// TIA Portal V18 export
FUNCTION_BLOCK "FB2-meteringFB"   // FB2, LAD
{ S7_Optimized_Access := 'TRUE' }
VERSION : 0.1
// stored: AutoNumber true, IsIECCheckEnabled false, IsRetainMemResEnabled false, MemoryReserve 100, SetENOAutomatically false, UDAEnableTagReadback false
   VAR_INPUT
      Metering_function : Int;
      "DO Continuous metering" : Bool;
      Dispensing_time : DInt;
      "Set Qty in ml" : Real;
      "VC1 Pulses" : DInt;
      "VC2 Pulses" : DInt;
      VC1_impulse : Real;
      VC2_impulse : Real;
      "Outlet Open  to Pump ON A delay" : DInt;
      "Outlet Open  to Pump ON B delay" : DInt;
      "Pump Off  to Inlet A Close" : DInt;
      "Pump Off  to Inlet B Close" : DInt;
      "Mixer ON to Outlet ON" : DInt;
      "Pump Off  to Outlet Close" : DInt;
      "Outlet Close to Mixer Off" : DInt;
   END_VAR
   VAR_OUTPUT
      "Volume dispensed" : Real;
      "Run time" : Int;
   END_VAR
   VAR_IN_OUT
      ON_inlet_A : Bool;
      ON_inlet_B : Bool;
      ON_Pump_A : Bool;
      ON_pump_B : Bool;
      ON_valve_A : Bool;
      ON_valve_B : Bool;
      ON_Mixer : Bool;
      "Start Metering" : Bool;
      "Stop metering" : Bool;
      "Process running" : Bool;
      "process completed" : Bool;
   END_VAR
   VAR
      "pump A to valveA delay" : Bool;
      "Pump B to valve B delay" : Bool;
      "Pump Off to mixer off delay_1" : Bool;
      "VC1 pulses prev" : DInt;
      "VC2 pulses prev" : DInt;
      "VC1 pulse generted" : DInt;
      "VC2 pulse generated" : DInt;
      "Pump A Voulme dispensed" : Real;
      "Pump B volume dispensed" : Real;
      "Total Volume dispensed" : Real;
      "metering started" : Bool;
      "metering time in msec" : DInt;
      "dispense time elapsed" : Bool;
      R_TRIG_Instance { S7_SetPoint := 'True'} : R_TRIG;
      IEC_Timer_0_Instance { S7_SetPoint := 'True'} : TON_TIME;
      IEC_Timer_0_Instance_1 { S7_SetPoint := 'True'} : TON_TIME;
      IEC_Timer_0_Instance_2 { S7_SetPoint := 'True'} : TON_TIME;
      R_TRIG_Instance_1 { S7_SetPoint := 'True'} : R_TRIG;
      temp { S7_SetPoint := 'True'} : Bool;
      IEC_Timer_0_Instance_3 { S7_SetPoint := 'True'} : TON_TIME;
      IEC_Timer_0_Instance_4 { S7_SetPoint := 'True'} : TON_TIME;
      IEC_Timer_0_Instance_5 { S7_SetPoint := 'True'} : TON_TIME;
      IEC_Timer_0_Instance_6 { S7_SetPoint := 'True'} : TON_TIME;
      IEC_Timer_0_Instance_7 { S7_SetPoint := 'True'} : TON_TIME;
      IEC_Timer_0_Instance_8 { S7_SetPoint := 'True'} : TON_TIME;
   END_VAR
   VAR_TEMP
      Ons_temp : Bool;
   END_VAR
   VAR_TEMP   // added for the SCL form of the ladder/FBD networks
      _w1 : Bool;
      _w2 : Bool;
      _w3 : Bool;
   END_VAR
BEGIN

REGION Network 1
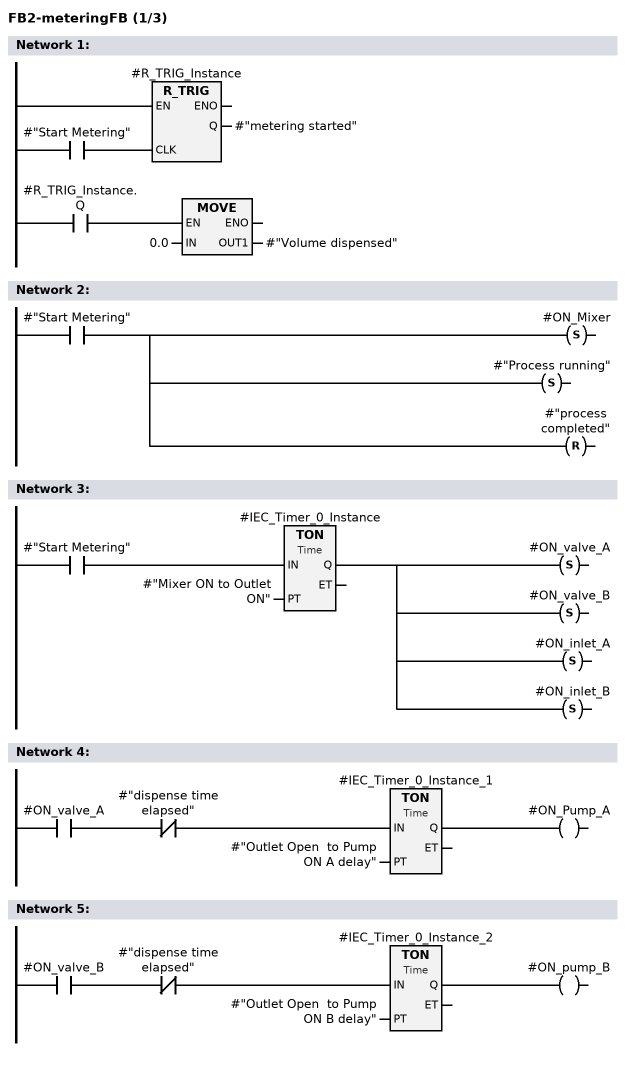
   RUNG wire#powerrail
      #R_TRIG_Instance.R_TRIG(CLK := wire#w1, Q => #"metering started")
   END_RUNG
   RUNG wire#powerrail
      Contact( #"Start Metering" )
   END_RUNG wire#w1
   RUNG wire#powerrail
      Contact( #R_TRIG_Instance.Q )
      Move(in := 0.0, out1 => #"Volume dispensed")
   END_RUNG
   // the same network as SCL:
   #R_TRIG_Instance(CLK := #"Start Metering", Q => #"metering started");   // R_TRIG
   IF #R_TRIG_Instance.Q THEN #"Volume dispensed" := 0.0; END_IF;
END_REGION

REGION Network 2
   RUNG wire#powerrail
      Contact( #"Start Metering" )
      wire#w1
      S_Coil( #ON_Mixer )
   END_RUNG
   RUNG wire#w1
      S_Coil( #"Process running" )
   END_RUNG
   RUNG wire#w1
      R_Coil( #"process completed" )
   END_RUNG
   // the same network as SCL:
   IF #"Start Metering" THEN
       #ON_Mixer := TRUE;
       #"Process running" := TRUE;
       #"process completed" := FALSE;
   END_IF;
END_REGION

REGION Network 3
   RUNG wire#powerrail
      Contact( #"Start Metering" )
      { S7_Templates := "time_type := Time" } #IEC_Timer_0_Instance.TON(pt := #"Mixer ON to Outlet ON", et =>)
      wire#w1
      S_Coil( #ON_valve_A )
   END_RUNG
   RUNG wire#w1
      S_Coil( #ON_valve_B )
   END_RUNG
   RUNG wire#w1
      S_Coil( #ON_inlet_A )
   END_RUNG
   RUNG wire#w1
      S_Coil( #ON_inlet_B )
   END_RUNG
   // the same network as SCL:
   #IEC_Timer_0_Instance(IN := #"Start Metering", PT := #"Mixer ON to Outlet ON");   // TON
   IF #IEC_Timer_0_Instance.Q THEN
       #ON_valve_A := TRUE;
       #ON_valve_B := TRUE;
       #ON_inlet_A := TRUE;
       #ON_inlet_B := TRUE;
   END_IF;
END_REGION

REGION Network 4
   RUNG wire#powerrail
      Contact( #ON_valve_A )
      I_Contact( #"dispense time elapsed" )
      { S7_Templates := "time_type := Time" } #IEC_Timer_0_Instance_1.TON(pt := #"Outlet Open  to Pump ON A delay", et =>)
      Coil( #ON_Pump_A )
   END_RUNG
   // the same network as SCL:
   #IEC_Timer_0_Instance_1(IN := #ON_valve_A AND NOT #"dispense time elapsed",   // TON
                           PT := #"Outlet Open  to Pump ON A delay");
   #ON_Pump_A := #IEC_Timer_0_Instance_1.Q;
END_REGION

REGION Network 5
   RUNG wire#powerrail
      Contact( #ON_valve_B )
      I_Contact( #"dispense time elapsed" )
      { S7_Templates := "time_type := Time" } #IEC_Timer_0_Instance_2.TON(pt := #"Outlet Open  to Pump ON B delay", et =>)
      Coil( #ON_pump_B )
   END_RUNG
   // the same network as SCL:
   #IEC_Timer_0_Instance_2(IN := #ON_valve_B AND NOT #"dispense time elapsed",   // TON
                           PT := #"Outlet Open  to Pump ON B delay");
   #ON_pump_B := #IEC_Timer_0_Instance_2.Q;
END_REGION

REGION Network 6
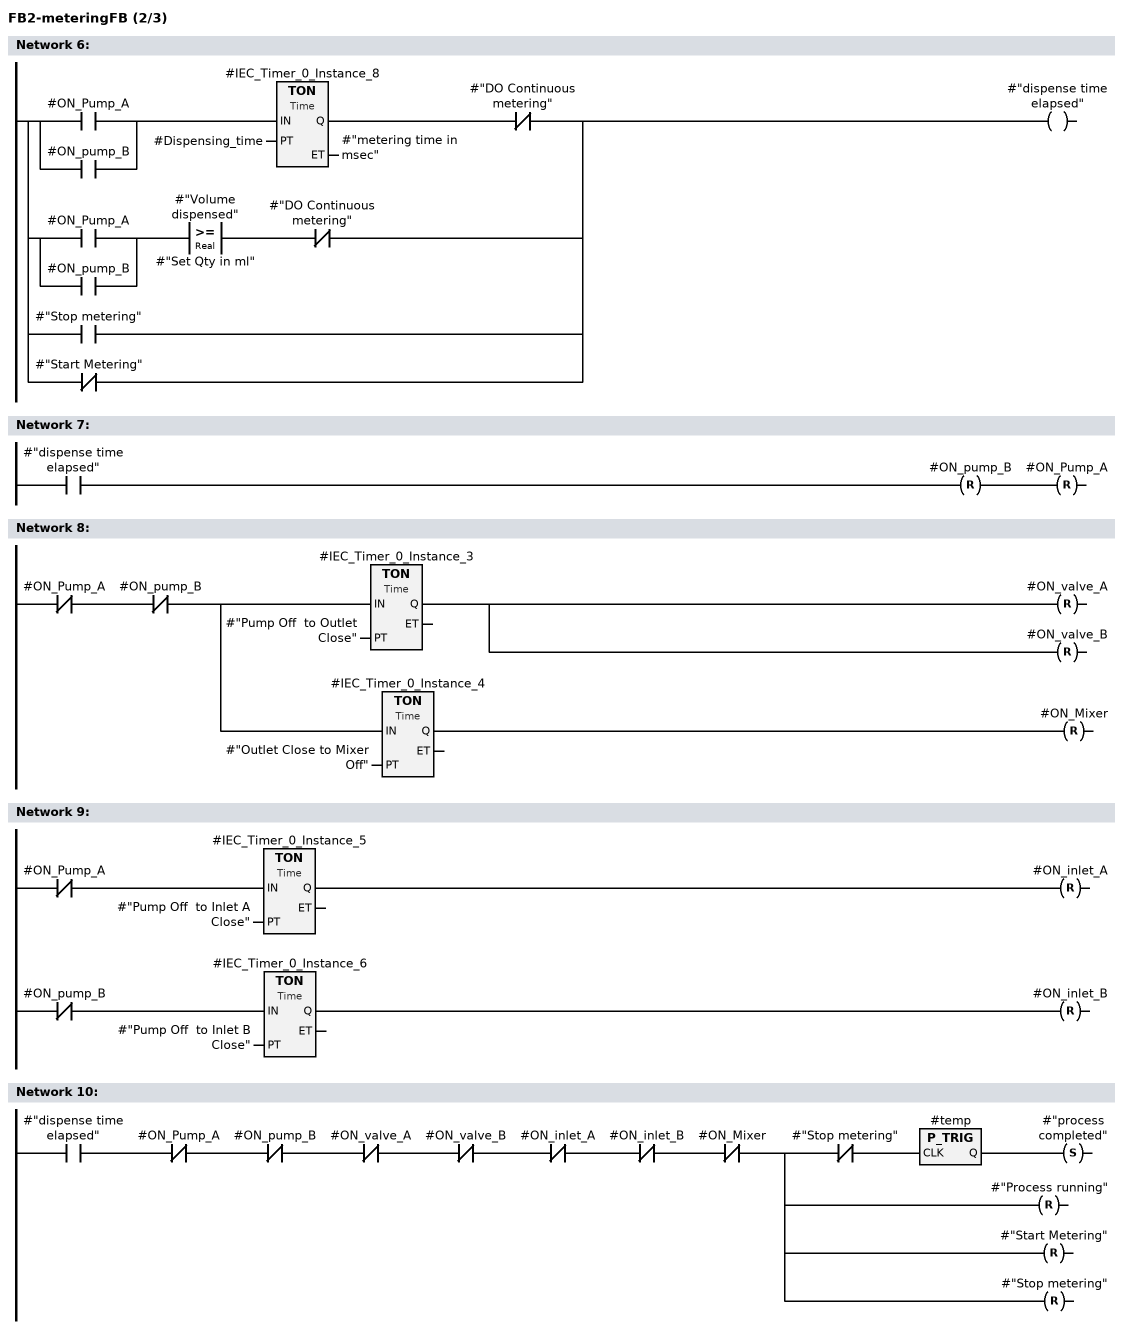
   RUNG wire#powerrail
      Contact( #ON_Pump_A )
      wire#w1
      { S7_Templates := "time_type := Time" } #IEC_Timer_0_Instance_8.TON(pt := #Dispensing_time, et => #"metering time in msec")
      I_Contact( #"DO Continuous metering" )
      wire#w2
      Coil( #"dispense time elapsed" )
   END_RUNG
   RUNG wire#powerrail
      Contact( #ON_pump_B )
   END_RUNG wire#w1
   RUNG wire#powerrail
      Contact( #ON_Pump_A )
      wire#w3
      { S7_Templates := "SrcType := Real" } GE_Contact(in1 := #"Volume dispensed", in2 := #"Set Qty in ml")
      I_Contact( #"DO Continuous metering" )
   END_RUNG wire#w2
   RUNG wire#powerrail
      Contact( #ON_pump_B )
   END_RUNG wire#w3
   RUNG wire#powerrail
      Contact( #"Stop metering" )
   END_RUNG wire#w2
   RUNG wire#powerrail
      I_Contact( #"Start Metering" )
   END_RUNG wire#w2
   // the same network as SCL:
   #IEC_Timer_0_Instance_8(IN := #ON_Pump_A OR #ON_pump_B,   // TON
                           PT := #Dispensing_time,
                           ET => #"metering time in msec");
   #"dispense time elapsed" := (#IEC_Timer_0_Instance_8.Q AND NOT #"DO Continuous metering") OR ((#ON_Pump_A OR #ON_pump_B) AND (#"Volume dispensed" >= #"Set Qty in ml") AND NOT #"DO Continuous metering") OR #"Stop metering" OR NOT #"Start Metering";
END_REGION

REGION Network 7
   RUNG wire#powerrail
      Contact( #"dispense time elapsed" )
      R_Coil( #ON_pump_B )
      R_Coil( #ON_Pump_A )
   END_RUNG
   // the same network as SCL:
   IF #"dispense time elapsed" THEN
       #ON_pump_B := FALSE;
       #ON_Pump_A := FALSE;
   END_IF;
END_REGION

REGION Network 8
   RUNG wire#powerrail
      I_Contact( #ON_Pump_A )
      I_Contact( #ON_pump_B )
      wire#w1
      { S7_Templates := "time_type := Time" } #IEC_Timer_0_Instance_3.TON(pt := #"Pump Off  to Outlet Close", et =>)
      wire#w2
      R_Coil( #ON_valve_A )
   END_RUNG
   RUNG wire#w2
      R_Coil( #ON_valve_B )
   END_RUNG
   RUNG wire#w1
      { S7_Templates := "time_type := Time" } #IEC_Timer_0_Instance_4.TON(pt := #"Outlet Close to Mixer Off", et =>)
      R_Coil( #ON_Mixer )
   END_RUNG
   // the same network as SCL:
   #_w1 := NOT #ON_Pump_A AND NOT #ON_pump_B;
   #IEC_Timer_0_Instance_3(IN := #_w1, PT := #"Pump Off  to Outlet Close");   // TON
   IF #IEC_Timer_0_Instance_3.Q THEN
       #ON_valve_A := FALSE;
       #ON_valve_B := FALSE;
   END_IF;
   #IEC_Timer_0_Instance_4(IN := #_w1, PT := #"Outlet Close to Mixer Off");   // TON
   IF #IEC_Timer_0_Instance_4.Q THEN #ON_Mixer := FALSE; END_IF;
END_REGION

REGION Network 9
   RUNG wire#powerrail
      I_Contact( #ON_Pump_A )
      { S7_Templates := "time_type := Time" } #IEC_Timer_0_Instance_5.TON(pt := #"Pump Off  to Inlet A Close", et =>)
      R_Coil( #ON_inlet_A )
   END_RUNG
   RUNG wire#powerrail
      I_Contact( #ON_pump_B )
      { S7_Templates := "time_type := Time" } #IEC_Timer_0_Instance_6.TON(pt := #"Pump Off  to Inlet B Close", et =>)
      R_Coil( #ON_inlet_B )
   END_RUNG
   // the same network as SCL:
   #IEC_Timer_0_Instance_5(IN := NOT #ON_Pump_A, PT := #"Pump Off  to Inlet A Close");   // TON
   IF #IEC_Timer_0_Instance_5.Q THEN #ON_inlet_A := FALSE; END_IF;
   #IEC_Timer_0_Instance_6(IN := NOT #ON_pump_B, PT := #"Pump Off  to Inlet B Close");   // TON
   IF #IEC_Timer_0_Instance_6.Q THEN #ON_inlet_B := FALSE; END_IF;
END_REGION

REGION Network 10
   RUNG wire#powerrail
      Contact( #"dispense time elapsed" )
      I_Contact( #ON_Pump_A )
      I_Contact( #ON_pump_B )
      I_Contact( #ON_valve_A )
      I_Contact( #ON_valve_B )
      I_Contact( #ON_inlet_A )
      I_Contact( #ON_inlet_B )
      I_Contact( #ON_Mixer )
      wire#w1
      I_Contact( #"Stop metering" )
      P_Trig( #temp )
      S_Coil( #"process completed" )
   END_RUNG
   RUNG wire#w1
      R_Coil( #"Process running" )
   END_RUNG
   RUNG wire#w1
      R_Coil( #"Start Metering" )
   END_RUNG
   RUNG wire#w1
      R_Coil( #"Stop metering" )
   END_RUNG
   // the same network as SCL:
   #_w1 := #"dispense time elapsed" AND NOT #ON_Pump_A AND NOT #ON_pump_B AND NOT #ON_valve_A AND NOT #ON_valve_B AND NOT #ON_inlet_A AND NOT #ON_inlet_B AND NOT #ON_Mixer;
   #_w2 := #_w1 AND NOT #"Stop metering";
   #_w3 := #_w2 AND NOT #temp;   // rising edge
   #temp := #_w2;
   IF #_w3 THEN #"process completed" := TRUE; END_IF;
   IF #_w1 THEN
       #"Process running" := FALSE;
       #"Start Metering" := FALSE;
       #"Stop metering" := FALSE;
   END_IF;
END_REGION

REGION Network 11
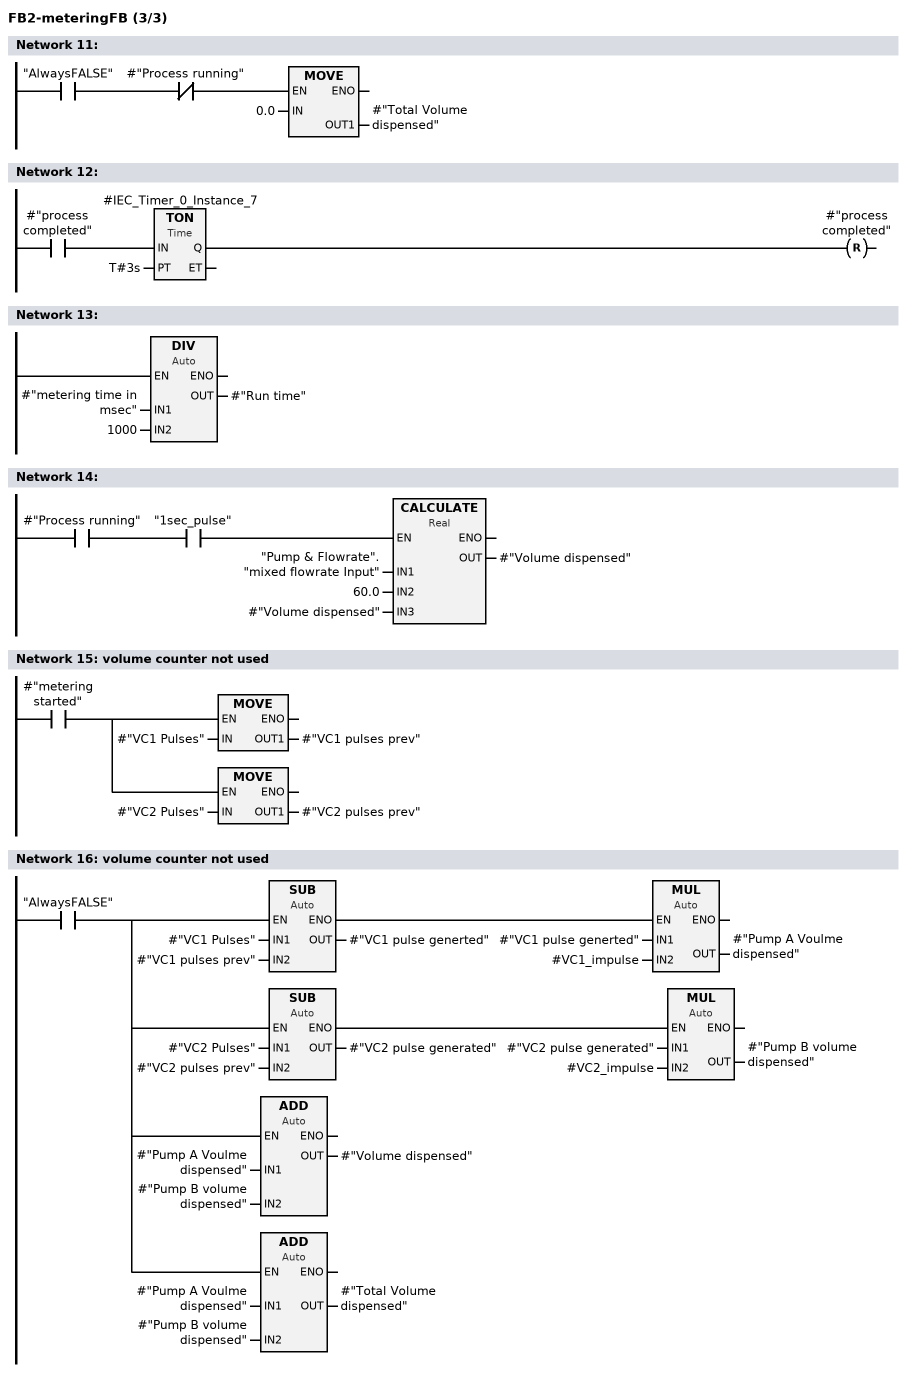
   RUNG wire#powerrail
      Contact( "AlwaysFALSE" )
      I_Contact( #"Process running" )
      Move(in := 0.0, out1 => #"Total Volume dispensed")
   END_RUNG
   // the same network as SCL:
   IF "AlwaysFALSE" AND NOT #"Process running" THEN #"Total Volume dispensed" := 0.0; END_IF;
END_REGION

REGION Network 12
   RUNG wire#powerrail
      Contact( #"process completed" )
      { S7_Templates := "time_type := Time" } #IEC_Timer_0_Instance_7.TON(pt := T#3s, et =>)
      R_Coil( #"process completed" )
   END_RUNG
   // the same network as SCL:
   #IEC_Timer_0_Instance_7(IN := #"process completed", PT := T#3s);   // TON
   IF #IEC_Timer_0_Instance_7.Q THEN #"process completed" := FALSE; END_IF;
END_REGION

REGION Network 13
   RUNG wire#powerrail
      Div(in1 := #"metering time in msec", in2 := 1000, out => #"Run time")
   END_RUNG
   // the same network as SCL:
   #"Run time" := #"metering time in msec" / 1000;
END_REGION

REGION Network 14
   RUNG wire#powerrail
      Contact( #"Process running" )
      Contact( "1sec_pulse" )
      { S7_Templates := "SrcType := Real"; S7_Expression := "(IN1/IN2)+IN3" } Calculate(in1 := "Pump & Flowrate"."mixed flowrate Input", in2 := 60.0, in3 := #"Volume dispensed", out => #"Volume dispensed")
   END_RUNG
   // the same network as SCL:
   IF #"Process running" AND "1sec_pulse" THEN
       #"Volume dispensed" := ("Pump & Flowrate"."mixed flowrate Input"/60.0)+#"Volume dispensed";
   END_IF;
END_REGION

REGION Network 15: volume counter not used
   RUNG wire#powerrail
      Contact( #"metering started" )
      wire#w1
      Move(in := #"VC1 Pulses", out1 => #"VC1 pulses prev")
   END_RUNG
   RUNG wire#w1
      Move(in := #"VC2 Pulses", out1 => #"VC2 pulses prev")
   END_RUNG
   // the same network as SCL:
   IF #"metering started" THEN
       #"VC1 pulses prev" := #"VC1 Pulses";
       #"VC2 pulses prev" := #"VC2 Pulses";
   END_IF;
END_REGION

REGION Network 16: volume counter not used
   RUNG wire#powerrail
      Contact( "AlwaysFALSE" )
      wire#w1
      Sub(in1 := #"VC1 Pulses", in2 := #"VC1 pulses prev", out => #"VC1 pulse generted")
      Mul(in1 := #"VC1 pulse generted", in2 := #VC1_impulse, out => #"Pump A Voulme dispensed")
   END_RUNG
   RUNG wire#w1
      Sub(in1 := #"VC2 Pulses", in2 := #"VC2 pulses prev", out => #"VC2 pulse generated")
      Mul(in1 := #"VC2 pulse generated", in2 := #VC2_impulse, out => #"Pump B volume dispensed")
   END_RUNG
   RUNG wire#w1
      Add(in1 := #"Pump A Voulme dispensed", in2 := #"Pump B volume dispensed", out => #"Volume dispensed")
   END_RUNG
   RUNG wire#w1
      Add(in1 := #"Pump A Voulme dispensed", in2 := #"Pump B volume dispensed", out => #"Total Volume dispensed")
   END_RUNG
   // the same network as SCL:
   IF "AlwaysFALSE" THEN
       #"VC1 pulse generted" := #"VC1 Pulses" - #"VC1 pulses prev";
       #"Pump A Voulme dispensed" := #"VC1 pulse generted" * #VC1_impulse;
       #"VC2 pulse generated" := #"VC2 Pulses" - #"VC2 pulses prev";
       #"Pump B volume dispensed" := #"VC2 pulse generated" * #VC2_impulse;
       #"Volume dispensed" := #"Pump A Voulme dispensed" + #"Pump B volume dispensed";
       #"Total Volume dispensed" := #"Pump A Voulme dispensed" + #"Pump B volume dispensed";
   END_IF;
END_REGION
END_FUNCTION_BLOCK
